// TIA Portal V15.1 export
// export: Created 2024-05-17T05:38:21.5836216Z, ExportSetting WithDefaults, DisplayName Totally Integrated Automation Portal, DisplayVersion V15.1 Update 5, DisplayName TIA Portal Openness, DisplayVersion V15.1 Update 5, DisplayName SINAMICS Startdrive Advanced, DisplayVersion V15.1, DisplayName G130, G150, S120, S150, SINAMICS MV, S210, DisplayVersion V15.1, DisplayName G110M, G120, G120C, G120D, G120P, DisplayVersion V15.1, DisplayName STEP 7 Professional, DisplayVersion V15.1 Update 5, DisplayName STEP 7 Safety, DisplayVersion V15.1, DisplayName WinCC Professional, DisplayVersion V15.1 Update 5, DisplayName SIMATIC Visualization Architect, DisplayVersion V15.1
DATA_BLOCK "_209230ZS01Safety"   // DB425
{ S7_Optimized_Access := 'FALSE' }
VERSION : 0.1
// stored: AutoNumber false, DBAccessibleFromOPCUA true, IsOnlyStoredInLoadMemory false, IsWriteProtectedInAS false
   VAR RETAIN
      AA_209230AS10F9SH1 { ExternalAccessible := 'False'; ExternalVisible := 'False'; ExternalWritable := 'False'} : Bool;   // Emergency Stop push button 230AS10 (Operator panel)
      AA_209230AS30F9SH1 { ExternalAccessible := 'False'; ExternalVisible := 'False'; ExternalWritable := 'False'} : Bool;   // Emergency Stop push button 230AS30 (Light Beam panel)
      AA_209230ASD01F9SH1 { ExternalAccessible := 'False'; ExternalVisible := 'False'; ExternalWritable := 'False'} : Bool;   // Emergency Stop push button 230ASD01 (MGB)
      AA_209230ASH01F9SH1 { ExternalAccessible := 'False'; ExternalVisible := 'False'; ExternalWritable := 'False'} : Bool;   // Emergency Stop push button 230ASH01 (Handheld panel)
      AA_209230ASH01F9SH2 { ExternalAccessible := 'False'; ExternalVisible := 'False'; ExternalWritable := 'False'} : Bool;   // Deathmans switch 230ASH01 (Handheld panel)
      AA_209F9K13FB { ExternalAccessible := 'False'; ExternalVisible := 'False'; ExternalWritable := 'False'} : Bool;   // Feedback Alarm 212D R230.03/04 400VAC OFF
      AA_209230ASD01F9SG1 { ExternalAccessible := 'False'; ExternalVisible := 'False'; ExternalWritable := 'False'} : Bool;   // Safety Gate Switch Alarm 230ASD01 (MGB)
      AC_209230ASD01F9SG1EnablingSwitch { ExternalAccessible := 'False'; ExternalVisible := 'False'; ExternalWritable := 'False'} : Bool;   // Enabling Switch Connected 230ASD01 (MGB)
      AC_209230ASD01F9SG1Solenoid { ExternalAccessible := 'False'; ExternalVisible := 'False'; ExternalWritable := 'False'} : Bool;   // Solenoid Safety Gate Alarm 230ASD01 (MGB)
      AC_209230ASD01F9SG1AccesReq { ExternalAccessible := 'False'; ExternalVisible := 'False'; ExternalWritable := 'False'} : Bool;   // Acces Request Safety Gate 230ASD01 (MGB)
      AD_209230ASD01F9SG1DiagWarning { ExternalAccessible := 'False'; ExternalVisible := 'False'; ExternalWritable := 'False'} : Bool;   // Diagnostic Warning Safety Gate 230ASD01 (MGB)
      AA_209230AS10XS10 { ExternalAccessible := 'False'; ExternalVisible := 'False'; ExternalWritable := 'False'} : Bool;   // Dummy plug is missing, no Handheld is connected 230AS10 (Start/Stop panel)
      AA_209230ZS01SafetNotReseted { ExternalAccessible := 'False'; ExternalVisible := 'False'; ExternalWritable := 'False'} : Bool;   // Safety not Reseted 230ZS01
      AD_209230ZS01EmergencyStop { ExternalAccessible := 'False'; ExternalVisible := 'False'; ExternalWritable := 'False'} : Bool;   // Emergency Stop 230ZS01
      AD_209230ZS01GateStop { ExternalAccessible := 'False'; ExternalVisible := 'False'; ExternalWritable := 'False'} : Bool;   // Gate Stop 230ZS01
      AD_209230ZS01FbkError { ExternalAccessible := 'False'; ExternalVisible := 'False'; ExternalWritable := 'False'} : Bool;   // Feedback Error Pilz/Contactor 230ZS01
      AD_209230ZS01EStopPLC212 { ExternalAccessible := 'False'; ExternalVisible := 'False'; ExternalWritable := 'False'} : Bool;   // Emergency Stop from PLC212
      AD_209230ZS01MStopPLC212 { ExternalAccessible := 'False'; ExternalVisible := 'False'; ExternalWritable := 'False'} : Bool;   // Motion Stop from PLC212 for roller 230CA21
      AD_209230ZS01MStopPLC308 { ExternalAccessible := 'False'; ExternalVisible := 'False'; ExternalWritable := 'False'} : Bool;   // Motion Stop from PLC318 for roller 230CR22
      "230AS10F9SH1AlarmABCondition" { ExternalAccessible := 'False'; ExternalVisible := 'False'; ExternalWritable := 'False'} : Bool;   // Alarm AB Condition
      "230AS30F9SH1AlarmABCondition" { ExternalAccessible := 'False'; ExternalVisible := 'False'; ExternalWritable := 'False'} : Bool;   // Alarm AB Condition
      "230ASD01F9SH1AlarmABCondition" { ExternalAccessible := 'False'; ExternalVisible := 'False'; ExternalWritable := 'False'} : Bool;   // Alarm AB Condition
      "230ASH01F9SH1AlarmABCondition" { ExternalAccessible := 'False'; ExternalVisible := 'False'; ExternalWritable := 'False'} : Bool;   // Alarm AB Condition
      "230ASH01F9SH2AlarmABCondition" { ExternalAccessible := 'False'; ExternalVisible := 'False'; ExternalWritable := 'False'} : Bool;   // Alarm AB Condition
      "209F9K13FBAlarmABCondition" { ExternalAccessible := 'False'; ExternalVisible := 'False'; ExternalWritable := 'False'} : Bool;   // Alarm AB Condition
      "230AS10XS10AlarmABCondition" { ExternalAccessible := 'False'; ExternalVisible := 'False'; ExternalWritable := 'False'} : Bool;   // Alarm AB Condition
      SafetyNotResetedAlarmABCondition { ExternalAccessible := 'False'; ExternalVisible := 'False'; ExternalWritable := 'False'} : Bool;   // Alarm AB Condition
      H_209230AS10F9SH1IAnim : Word;   // Icon Animation
      H_209230AS30F9SH1IAnim : Word;   // Icon Animation
      H_209230ASD01F9SH1IAnim : Word;   // Icon Animation
      H_209230ASH01F9SH1IAnim : Word;   // Icon Animation
      H_209230ASH01F9SH2IAnim : Word;   // Icon Animation
      H_209230ZS01F9SG1IAnim : Word;   // Icon Animation
      H_209F9K13FBIAnim : Word;   // Icon Animation
      H_209230AS10XS10IAnim : Word;   // Icon Animation
      H_209230ZS01SafetyNotResetedIAnim : Word;   // Icon Animation
      H_209230ZS01GateStopIAnim : Word;   // Icon Animation
      H_209230ZS01EmergencyStopIAnim : Word;   // Icon Animation
      H_209230ZS01FbkErrorIAnim : Word;   // Icon Animation
      H_209230ZS01EStopPLC212IAnim : Word;   // Icon Animation
      H_209230ZS01MStopPLC212IAnim : Word;   // Icon Animation
      H_209230ZS01MStopPLC308IAnim : Word;   // Icon Animation
      H_209230ZS01PassivIAnim : Word;   // Icon Animation
      H_Anim : Word;   // Animation
      H_DBnr : Int;   // DB number
      H : Struct   // HMI Animation
         "209230ASD01" : "H_GateLock-MGB-Maint";   // HMI Animation
      END_STRUCT;
      H_HMI : Struct   // HMI Animation
         "209230ASD01" : "H_HMI";   // HMI Animation
      END_STRUCT;
      "209230ASD01" { ExternalAccessible := 'False'; ExternalVisible := 'False'; ExternalWritable := 'False'} : "MGB";   // MGB Gate Lock
      "230ZS01F9SG1" { ExternalAccessible := 'False'; ExternalVisible := 'False'; ExternalWritable := 'False'} : "AlarmBits";   // Alarm Bits
      Passivation { ExternalAccessible := 'False'; ExternalVisible := 'False'; ExternalWritable := 'False'} : "AlarmBits";   // Passivation Alarm Bits / Alarm A
      AlarmA { ExternalAccessible := 'False'; ExternalVisible := 'False'; ExternalWritable := 'False'} : Bool;   // Alarm A
      AlarmB { ExternalAccessible := 'False'; ExternalVisible := 'False'; ExternalWritable := 'False'} : Bool;   // Alarm B
      AlarmC { ExternalAccessible := 'False'; ExternalVisible := 'False'; ExternalWritable := 'False'} : Bool;   // Alarm C
      AlarmD { ExternalAccessible := 'False'; ExternalVisible := 'False'; ExternalWritable := 'False'} : Bool;   // Alarm D
      AlarmABCondition { ExternalAccessible := 'False'; ExternalVisible := 'False'; ExternalWritable := 'False'} : Bool;   // Summary Alarm AB condition
      SafetyObjectAckReq230AS10 { ExternalAccessible := 'False'; ExternalVisible := 'False'; ExternalWritable := 'False'} : Bool;   // Safety Status ACK REQ
      SafetyObjectAckReq230AS30 { ExternalAccessible := 'False'; ExternalVisible := 'False'; ExternalWritable := 'False'} : Bool;   // Safety Status ACK REQ
      SafetyObjectAckReq230ASD01 { ExternalAccessible := 'False'; ExternalVisible := 'False'; ExternalWritable := 'False'} : Bool;   // Safety Status ACK REQ
      SafetyObjectAckReq230ASH01 { ExternalAccessible := 'False'; ExternalVisible := 'False'; ExternalWritable := 'False'} : Bool;   // Safety Status ACK REQ
      PowerOnRequest { ExternalAccessible := 'False'; ExternalVisible := 'False'; ExternalWritable := 'False'} : Bool;   // Power On Request
      ResetSafetyActive { ExternalAccessible := 'False'; ExternalVisible := 'False'; ExternalWritable := 'False'} : Bool;   // Reset Safety Active
      FeedbackError { ExternalAccessible := 'False'; ExternalVisible := 'False'; ExternalWritable := 'False'} : Bool;   // Feedback Error
      Check230AS10XS10 { ExternalAccessible := 'False'; ExternalVisible := 'False'; ExternalWritable := 'False'} : Bool;   // Check if dummy plug is ok
   END_VAR
BEGIN
END_DATA_BLOCK
